TYPE SetBrakeProcessArgs :
STRUCT
	///Requested brake state
	newState: DriveBrakeStates;
END_STRUCT
END_TYPE

(* stored: Version 1.1.0.1, ProductVersion 3.1.4019.2
   DUT SetBrakeProcessArgs: Id {2aa7961a-51c6-41fb-b707-78ad03af32d5} *)
